// TwinCAT 3 PLC project ProjectEuler
// Title: Project Euler
// Company: Open source
// Author: Open source contributers.
// ProjectVersion: 1.0.0
// Description: Open source project to solve Project euler problems with TwinCAT.
// ProgramVersion: 3.1.4023.0
// libraries:
//   Tc2_Standard, * (Beckhoff Automation GmbH)
//   Tc2_System, * (Beckhoff Automation GmbH)
//   Tc2_Utilities, * (Beckhoff Automation GmbH)
//   Tc3_Module, * (Beckhoff Automation GmbH)
//   TcUnit, * (www.tcunit.org)
// project tree:
//   / PlcTestTask.TcTTO
//   POUs/ PRG_TEST.TcPOU
//   POUs/Problems/Base/ FbProblemSolverBase.TcPOU, IProblemSolver.TcIO
//   POUs/Problems/ Problem1.TcPOU, Problem2.TcPOU, Problem3.TcPOU
//   POUs/Tests/ FbProblemTester.TcPOU

CONFIGURATION ProjectEuler
    RESOURCE PLC ON TwinCAT3
        TASK PlcTestTask(INTERVAL := T#10ms, PRIORITY := 20);
        PROGRAM PRG_TEST WITH PlcTestTask : PRG_TEST;
    END_RESOURCE
END_CONFIGURATION

// ---- POUs/Problems/Base/IProblemSolver.TcIO
INTERFACE IProblemSolver

{attribute 'monitoring' := 'call'}
PROPERTY Busy : BOOL
GET
END_GET
END_PROPERTY

METHOD Cyclic
VAR_INPUT
END_VAR
END_METHOD

{attribute 'monitoring' := 'call'}
PROPERTY Done : BOOL
GET
END_GET
END_PROPERTY

{attribute 'monitoring' := 'call'}
PROPERTY Execute : BOOL
GET
END_GET
SET
END_SET
END_PROPERTY

{attribute 'monitoring' := 'call'}
PROPERTY Result : String
GET
END_GET
END_PROPERTY

END_INTERFACE

// ---- POUs/PRG_TEST.TcPOU
PROGRAM PRG_TEST
VAR
    _problem1 : Problem1;
    _problem1Test : FbProblemTester(_problem1, '233168');
    _problem2 : Problem2;
    _problem2Test : FbProblemTester(_problem2, '4613732');
	_problem3 : Problem3;
	_problem3Test : FbProblemTester(_problem3, '6857');
END_VAR

TcUnit.RUN();

END_PROGRAM

// ---- POUs/Problems/Problem1.TcPOU
FUNCTION_BLOCK FINAL Problem1 EXTENDS FbProblemSolverBase

super^();

METHOD PROTECTED CyclicAction
VAR_OUTPUT
    complete : BOOL;
    result : STRING;
END_VAR
VAR
    _i : LINT;
    _sum : LINT;
END_VAR
(*Multiples OF 3 OR 5  
Problem 1
If we list all the natural numbers below 10 that are multiples of 3 or 5, we get 3, 5, 6 and 9. The sum of these multiples is 23.
Find the sum of all the multiples of 3 or 5 below 1000.*)
FOR _i := 0 TO 999 DO
    IF _i MOD 3 = 0 OR _i MOD 5 = 0 THEN
        _sum := _sum + _i;
    END_IF
END_FOR

result := LINT_TO_STRING(_sum);
complete := TRUE;
END_METHOD

END_FUNCTION_BLOCK

// ---- POUs/Problems/Base/FbProblemSolverBase.TcPOU
{attribute 'hide_all_locals'}
FUNCTION_BLOCK ABSTRACT FbProblemSolverBase IMPLEMENTS IProblemSolver
VAR
    _execute : BOOL;
    _busy : BOOL;
    _done : BOOL;
    _result : STRING;
    _state : (
        Idle,
        Executing,
        Resetting
    );

    _resetDoneOnFallingEdgeExecute : BOOL;
END_VAR
VAR_TEMP
    _again : BOOL;
    _complete : BOOL;
    _tempResult : STRING;
END_VAR

REPEAT
    _again := FALSE;

    CASE _state OF
        Idle:
            IF Execute THEN
                _state := _state + 1;
                _busy := TRUE;
                _done := FALSE;
                _again := TRUE;
            END_IF

        Executing:
            CyclicAction(complete => _complete, result => _tempResult);

            IF _complete THEN
                _state := _state + 1;
                _again := TRUE;
                _result := _tempResult;
                _busy := FALSE;
                _done := TRUE;
            END_IF

        Resetting:
            IF NOT Execute THEN
                ResetAction(complete => _complete);

                IF _resetDoneOnFallingEdgeExecute THEN
                    _done := FALSE;
                END_IF

                IF _complete THEN
                    _state := 0;
                    _again := TRUE;
                END_IF
            ELSE
                _resetDoneOnFallingEdgeExecute := TRUE;
            END_IF
    END_CASE
UNTIL NOT _again
END_REPEAT

{attribute 'monitoring' := 'call'}
PROPERTY PUBLIC Busy : BOOL
GET
Busy := _busy;
END_GET
END_PROPERTY

METHOD PUBLIC Cyclic
this^();
END_METHOD

METHOD PROTECTED ABSTRACT CyclicAction
VAR_OUTPUT
    complete : BOOL;
    result : STRING;
END_VAR
END_METHOD

{attribute 'monitoring' := 'call'}
PROPERTY PUBLIC Done : BOOL
GET
Done := _done;
END_GET
END_PROPERTY

{attribute 'monitoring' := 'call'}
PROPERTY Execute : BOOL
GET
Execute := _execute;
END_GET
SET
_execute := Execute;
END_SET
END_PROPERTY

METHOD PROTECTED ResetAction
VAR_OUTPUT
    complete : BOOL;
END_VAR
complete := true;
END_METHOD

{attribute 'monitoring' := 'call'}
PROPERTY PUBLIC Result : STRING
GET
Result := _result;
END_GET
END_PROPERTY

END_FUNCTION_BLOCK

// ---- POUs/Tests/FbProblemTester.TcPOU
FUNCTION_BLOCK FbProblemTester EXTENDS TcUnit.FB_TestSuite
VAR
    _problem : IProblemSolver;
    _expectedResult : STRING;
END_VAR

TEST(TestName := '');
_problem.Execute := TRUE;
_problem.Cyclic();

IF _problem.Done THEN
    AssertEquals_STRING(Expected := _expectedResult, Actual := _problem.Result, Message := 'The problem solver did not return the correct answer.');
    _problem.Execute := FALSE;
    TEST_FINISHED();
END_IF

METHOD FB_init : BOOL
VAR_INPUT
    bInitRetains : BOOL; // if TRUE, the retain variables are initialized (warm start / cold start)
    bInCopyCode : BOOL; // if TRUE, the instance afterwards gets moved into the copy code (online change)
    problemSolver : IProblemSolver;
    expectedResult : STRING;
END_VAR
_problem := problemSolver;
_expectedResult := expectedResult;
END_METHOD

END_FUNCTION_BLOCK

// ---- POUs/Problems/Problem2.TcPOU
FUNCTION_BLOCK FINAL Problem2 EXTENDS FbProblemSolverBase

super^();

METHOD PROTECTED CyclicAction
VAR_OUTPUT
    complete : BOOL;
    result : STRING;
END_VAR
VAR
    _term1 : LINT;
    _term2 : LINT := 1;
    _term3 : LINT;
    _sum : LINT;
END_VAR
(*Even Fibonacci numbers  
Problem 2
Each new term in the Fibonacci sequence is generated by adding the previous two terms. By starting with 1 and 2, the first 10 terms will be:
1, 2, 3, 5, 8, 13, 21, 34, 55, 89, ...
By considering the terms in the Fibonacci sequence whose values do not exceed four million, find the sum of the even-valued terms.
*)
WHILE TRUE DO
    _term3 := _term1 + _term2;

    IF _term3 > 4000000 THEN
        EXIT;
    ELSIF _term3 MOD 2 = 0 THEN
        _sum := _sum + _term3;
    END_IF

    _term1 := _term2;
    _term2 := _term3;
END_WHILE

result := LINT_TO_STRING(_sum);
complete := TRUE;
END_METHOD

END_FUNCTION_BLOCK

// ---- POUs/Problems/Problem3.TcPOU
FUNCTION_BLOCK FINAL Problem3 EXTENDS FbProblemSolverBase

super^();

METHOD PROTECTED  CyclicAction
VAR_OUTPUT
    complete : BOOL;
    result : STRING;
END_VAR
VAR
	_maxPrime : ULINT := 0;
	_n : ULINT := 600851475143;
	_i : ULINT := 5;
END_VAR
(*Largest prime factor
Problem 3
The prime factors of 13195 are 5, 7, 13 and 29.
What is the largest prime factor of the number 600851475143 ?
*)

WHILE _n MOD 2 = 0 DO
	_maxPrime := 2;
	_n := _n/2;
END_WHILE

WHILE _n MOD 3 = 0 DO
	_maxPrime := 3;
	_n := _n/3;
END_WHILE

WHILE _i <= TO_ULINT(SQRT(TO_REAL(_n))) DO
	WHILE _n MOD _i = 0 DO
		_maxPrime := _i;
		_n := _n/_i;
	END_WHILE
	WHILE _n MOD (_i+2) = 0 DO
		_maxPrime := _i+2;
		_n := _n/(_i+2);
	END_WHILE
	_i := _i + 6;
END_WHILE

IF _n > 4 THEN
	_maxPrime := _n;
END_IF

result := ULINT_TO_STRING(_maxPrime);
complete := TRUE;
END_METHOD

END_FUNCTION_BLOCK
